// TIA Portal V20 export
DATA_BLOCK "MP109"   // DB311
// stored: MemoryReserve 100
BEGIN
END_DATA_BLOCK
